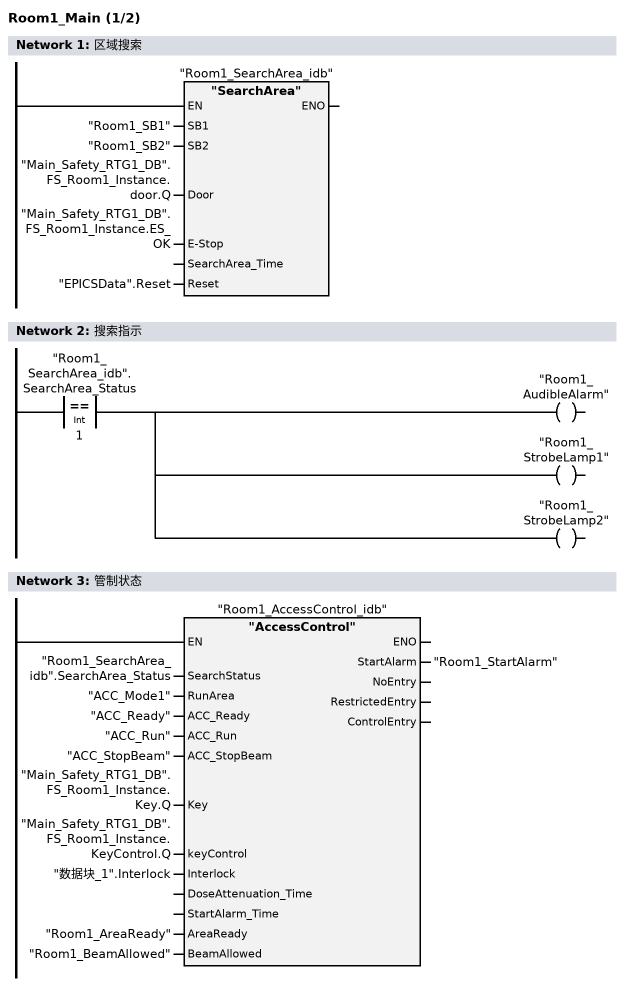
   RUNG wire#powerrail
      "Room1_SearchArea_idb"(SB1 := "Room1_SB1", SB2 := "Room1_SB2", Door := "Main_Safety_RTG1_DB".FS_Room1_Instance.door.Q, "E-Stop" := "Main_Safety_RTG1_DB".FS_Room1_Instance.ES_OK, SearchArea_Time :=, Reset := "EPICSData".Reset)
   END_RUNG
   // the same network as SCL:
   "Room1_SearchArea_idb"(SB1 := "Room1_SB1",   // "SearchArea"
                          SB2 := "Room1_SB2",
                          Door := "Main_Safety_RTG1_DB".FS_Room1_Instance.door.Q,
                          "E-Stop" := "Main_Safety_RTG1_DB".FS_Room1_Instance.ES_OK,
                          Reset := "EPICSData".Reset);
END_REGION

REGION Network 2: 搜索指示
   RUNG wire#powerrail
      { S7_Templates := "SrcType := Int" } EQ_Contact(in1 := "Room1_SearchArea_idb".SearchArea_Status, in2 := 1)
      wire#w1
      Coil( "Room1_AudibleAlarm" )
   END_RUNG
   RUNG wire#w1
      Coil( "Room1_StrobeLamp1" )
   END_RUNG
   RUNG wire#w1
      Coil( "Room1_StrobeLamp2" )
   END_RUNG
   // the same network as SCL:
   "Room1_AudibleAlarm" := "Room1_SearchArea_idb".SearchArea_Status = 1;
   "Room1_StrobeLamp1" := "Room1_AudibleAlarm";
   "Room1_StrobeLamp2" := "Room1_AudibleAlarm";
END_REGION

REGION Network 3: 管制状态
   RUNG wire#powerrail
      "Room1_AccessControl_idb"(SearchStatus := "Room1_SearchArea_idb".SearchArea_Status, RunArea := "ACC_Mode1", ACC_Ready := "ACC_Ready", ACC_Run := "ACC_Run", ACC_StopBeam := "ACC_StopBeam", Key := "Main_Safety_RTG1_DB".FS_Room1_Instance.Key.Q, keyControl := "Main_Safety_RTG1_DB".FS_Room1_Instance.KeyControl.Q, Interlock := "数据块_1".Interlock, DoseAttenuation_Time :=, StartAlarm_Time :=, AreaReady := "Room1_AreaReady", BeamAllowed := "Room1_BeamAllowed", StartAlarm => "Room1_StartAlarm", NoEntry =>, RestrictedEntry =>, ControlEntry =>)
   END_RUNG
   // the same network as SCL:
   "Room1_AccessControl_idb"(SearchStatus := "Room1_SearchArea_idb".SearchArea_Status,   // "AccessControl"
                           RunArea := "ACC_Mode1",
                           ACC_Ready := "ACC_Ready",
                           ACC_Run := "ACC_Run",
                           ACC_StopBeam := "ACC_StopBeam",
                           Key := "Main_Safety_RTG1_DB".FS_Room1_Instance.Key.Q,
                           keyControl := "Main_Safety_RTG1_DB".FS_Room1_Instance.KeyControl.Q,
                           Interlock := "数据块_1".Interlock,
                           AreaReady := "Room1_AreaReady",
                           BeamAllowed := "Room1_BeamAllowed",
                           StartAlarm => "Room1_StartAlarm");
END_REGION

REGION Network 4: 管制输出
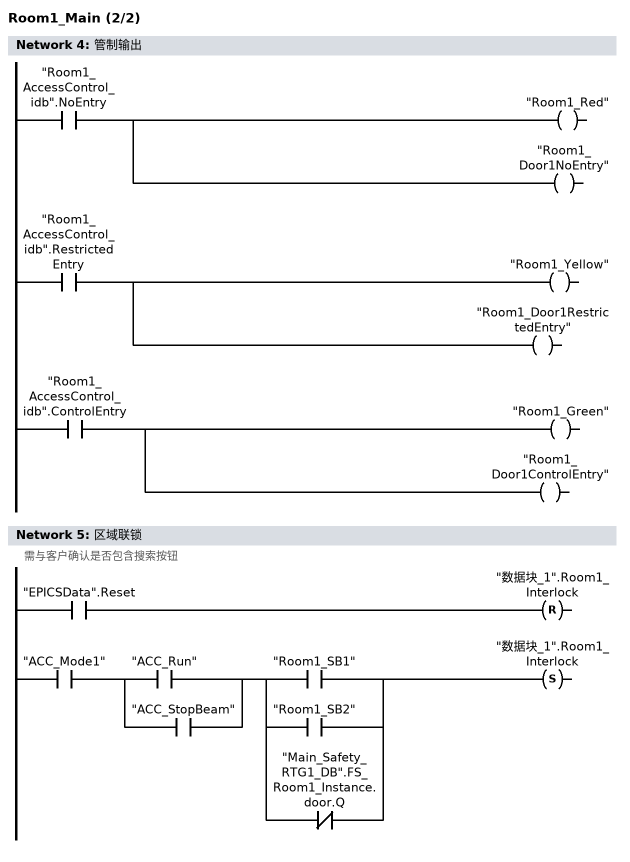
   RUNG wire#powerrail
      Contact( "Room1_AccessControl_idb".NoEntry )
      wire#w1
      Coil( "Room1_Red" )
   END_RUNG
   RUNG wire#w1
      Coil( "Room1_Door1NoEntry" )
   END_RUNG
   RUNG wire#powerrail
      Contact( "Room1_AccessControl_idb".RestrictedEntry )
      wire#w2
      Coil( "Room1_Yellow" )
   END_RUNG
   RUNG wire#w2
      Coil( "Room1_Door1RestrictedEntry" )
   END_RUNG
   RUNG wire#powerrail
      Contact( "Room1_AccessControl_idb".ControlEntry )
      wire#w3
      Coil( "Room1_Green" )
   END_RUNG
   RUNG wire#w3
      Coil( "Room1_Door1ControlEntry" )
   END_RUNG
   // the same network as SCL:
   "Room1_Red" := "Room1_AccessControl_idb".NoEntry;
   "Room1_Door1NoEntry" := "Room1_AccessControl_idb".NoEntry;
   "Room1_Yellow" := "Room1_AccessControl_idb".RestrictedEntry;
   "Room1_Door1RestrictedEntry" := "Room1_AccessControl_idb".RestrictedEntry;
   "Room1_Green" := "Room1_AccessControl_idb".ControlEntry;
   "Room1_Door1ControlEntry" := "Room1_AccessControl_idb".ControlEntry;
END_REGION

REGION Network 5: 区域联锁
   // 需与客户确认是否包含搜索按钮
   RUNG wire#powerrail
      Contact( "EPICSData".Reset )
      R_Coil( "数据块_1".Room1_Interlock )
   END_RUNG
   RUNG wire#powerrail
      Contact( "ACC_Mode1" )
      wire#w1
      Contact( "ACC_Run" )
      wire#w2
      Contact( "Room1_SB1" )
      wire#w3
      S_Coil( "数据块_1".Room1_Interlock )
   END_RUNG
   RUNG wire#w1
      Contact( "ACC_StopBeam" )
   END_RUNG wire#w2
   RUNG wire#w2
      Contact( "Room1_SB2" )
   END_RUNG wire#w3
   RUNG wire#w2
      I_Contact( "Main_Safety_RTG1_DB".FS_Room1_Instance.door.Q )
   END_RUNG wire#w3
   // the same network as SCL:
   IF "EPICSData".Reset THEN "数据块_1".Room1_Interlock := FALSE; END_IF;
   IF "ACC_Mode1" AND ("ACC_Run" OR "ACC_StopBeam") AND ("Room1_SB1" OR "Room1_SB2" OR NOT "Main_Safety_RTG1_DB".FS_Room1_Instance.door.Q) THEN
       "数据块_1".Room1_Interlock := TRUE;
   END_IF;
END_REGION
END_FUNCTION

FUNCTION "Room2_Main" : Void   // FC5, LAD
{ S7_Optimized_Access := 'TRUE' }
VERSION : 0.1
// stored: AutoNumber true, IsIECCheckEnabled false, SetENOAutomatically false, UDAEnableTagReadback false
BEGIN

REGION Network 1: 区域搜索
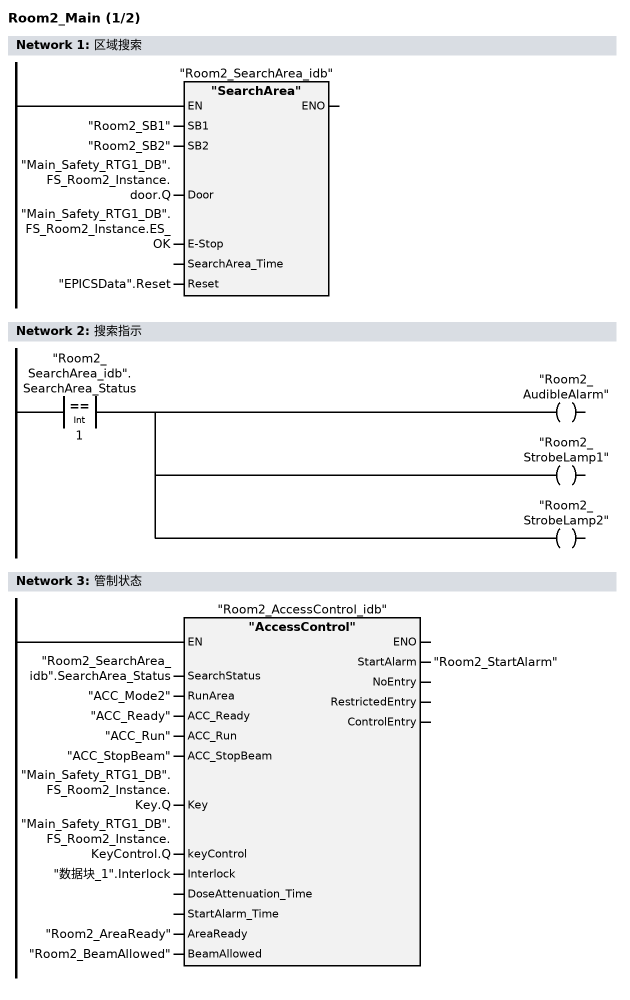
   RUNG wire#powerrail
      "Room2_SearchArea_idb"(SB1 := "Room2_SB1", SB2 := "Room2_SB2", Door := "Main_Safety_RTG1_DB".FS_Room2_Instance.door.Q, "E-Stop" := "Main_Safety_RTG1_DB".FS_Room2_Instance.ES_OK, SearchArea_Time :=, Reset := "EPICSData".Reset)
   END_RUNG
   // the same network as SCL:
   "Room2_SearchArea_idb"(SB1 := "Room2_SB1",   // "SearchArea"
                          SB2 := "Room2_SB2",
                          Door := "Main_Safety_RTG1_DB".FS_Room2_Instance.door.Q,
                          "E-Stop" := "Main_Safety_RTG1_DB".FS_Room2_Instance.ES_OK,
                          Reset := "EPICSData".Reset);
END_REGION

REGION Network 2: 搜索指示
   RUNG wire#powerrail
      { S7_Templates := "SrcType := Int" } EQ_Contact(in1 := "Room2_SearchArea_idb".SearchArea_Status, in2 := 1)
      wire#w1
      Coil( "Room2_AudibleAlarm" )
   END_RUNG
   RUNG wire#w1
      Coil( "Room2_StrobeLamp1" )
   END_RUNG
   RUNG wire#w1
      Coil( "Room2_StrobeLamp2" )
   END_RUNG
   // the same network as SCL:
   "Room2_AudibleAlarm" := "Room2_SearchArea_idb".SearchArea_Status = 1;
   "Room2_StrobeLamp1" := "Room2_AudibleAlarm";
   "Room2_StrobeLamp2" := "Room2_AudibleAlarm";
END_REGION

REGION Network 3: 管制状态
   RUNG wire#powerrail
      "Room2_AccessControl_idb"(SearchStatus := "Room2_SearchArea_idb".SearchArea_Status, RunArea := "ACC_Mode2", ACC_Ready := "ACC_Ready", ACC_Run := "ACC_Run", ACC_StopBeam := "ACC_StopBeam", Key := "Main_Safety_RTG1_DB".FS_Room2_Instance.Key.Q, keyControl := "Main_Safety_RTG1_DB".FS_Room2_Instance.KeyControl.Q, Interlock := "数据块_1".Interlock, DoseAttenuation_Time :=, StartAlarm_Time :=, AreaReady := "Room2_AreaReady", BeamAllowed := "Room2_BeamAllowed", StartAlarm => "Room2_StartAlarm", NoEntry =>, RestrictedEntry =>, ControlEntry =>)
   END_RUNG
   // the same network as SCL:
   "Room2_AccessControl_idb"(SearchStatus := "Room2_SearchArea_idb".SearchArea_Status,   // "AccessControl"
                           RunArea := "ACC_Mode2",
                           ACC_Ready := "ACC_Ready",
                           ACC_Run := "ACC_Run",
                           ACC_StopBeam := "ACC_StopBeam",
                           Key := "Main_Safety_RTG1_DB".FS_Room2_Instance.Key.Q,
                           keyControl := "Main_Safety_RTG1_DB".FS_Room2_Instance.KeyControl.Q,
                           Interlock := "数据块_1".Interlock,
                           AreaReady := "Room2_AreaReady",
                           BeamAllowed := "Room2_BeamAllowed",
                           StartAlarm => "Room2_StartAlarm");
END_REGION

REGION Network 4: 管制输出
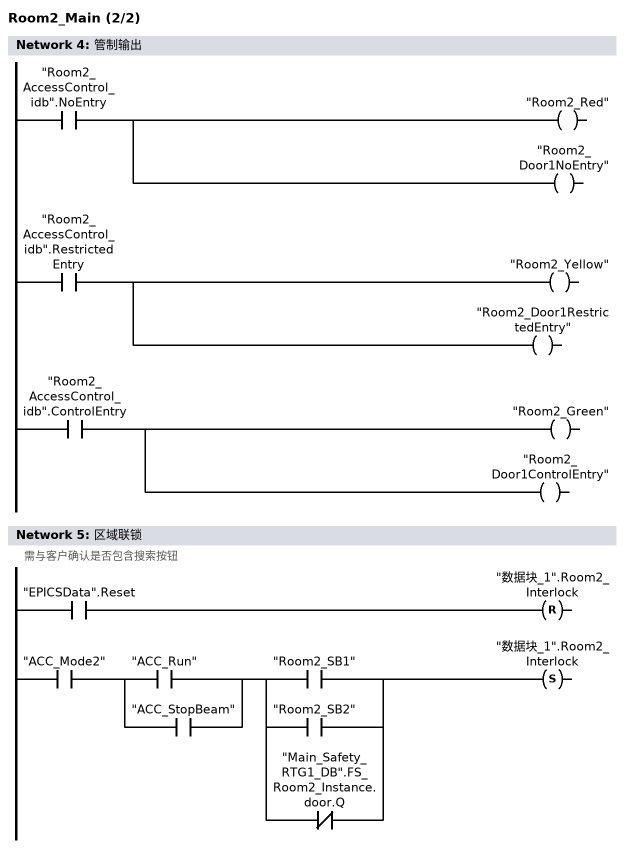
   RUNG wire#powerrail
      Contact( "Room2_AccessControl_idb".NoEntry )
      wire#w1
      Coil( "Room2_Red" )
   END_RUNG
   RUNG wire#w1
      Coil( "Room2_Door1NoEntry" )
   END_RUNG
   RUNG wire#powerrail
      Contact( "Room2_AccessControl_idb".RestrictedEntry )
      wire#w2
      Coil( "Room2_Yellow" )
   END_RUNG
   RUNG wire#w2
      Coil( "Room2_Door1RestrictedEntry" )
   END_RUNG
   RUNG wire#powerrail
      Contact( "Room2_AccessControl_idb".ControlEntry )
      wire#w3
      Coil( "Room2_Green" )
   END_RUNG
   RUNG wire#w3
      Coil( "Room2_Door1ControlEntry" )
   END_RUNG
   // the same network as SCL:
   "Room2_Red" := "Room2_AccessControl_idb".NoEntry;
   "Room2_Door1NoEntry" := "Room2_AccessControl_idb".NoEntry;
   "Room2_Yellow" := "Room2_AccessControl_idb".RestrictedEntry;
   "Room2_Door1RestrictedEntry" := "Room2_AccessControl_idb".RestrictedEntry;
   "Room2_Green" := "Room2_AccessControl_idb".ControlEntry;
   "Room2_Door1ControlEntry" := "Room2_AccessControl_idb".ControlEntry;
END_REGION

REGION Network 5: 区域联锁
   // 需与客户确认是否包含搜索按钮
   RUNG wire#powerrail
      Contact( "EPICSData".Reset )
      R_Coil( "数据块_1".Room2_Interlock )
   END_RUNG
   RUNG wire#powerrail
      Contact( "ACC_Mode2" )
      wire#w1
      Contact( "ACC_Run" )
      wire#w2
      Contact( "Room2_SB1" )
      wire#w3
      S_Coil( "数据块_1".Room2_Interlock )
   END_RUNG
   RUNG wire#w1
      Contact( "ACC_StopBeam" )
   END_RUNG wire#w2
   RUNG wire#w2
      Contact( "Room2_SB2" )
   END_RUNG wire#w3
   RUNG wire#w2
      I_Contact( "Main_Safety_RTG1_DB".FS_Room2_Instance.door.Q )
   END_RUNG wire#w3
   // the same network as SCL:
   IF "EPICSData".Reset THEN "数据块_1".Room2_Interlock := FALSE; END_IF;
   IF "ACC_Mode2" AND ("ACC_Run" OR "ACC_StopBeam") AND ("Room2_SB1" OR "Room2_SB2" OR NOT "Main_Safety_RTG1_DB".FS_Room2_Instance.door.Q) THEN
       "数据块_1".Room2_Interlock := TRUE;
   END_IF;
END_REGION
END_FUNCTION

FUNCTION "ACC_Main" : Void   // FC6, LAD
{ S7_Optimized_Access := 'TRUE' }
VERSION : 0.1
// stored: AutoNumber true, IsIECCheckEnabled false, SetENOAutomatically false, UDAEnableTagReadback false
BEGIN

REGION Network 1: 区域搜索
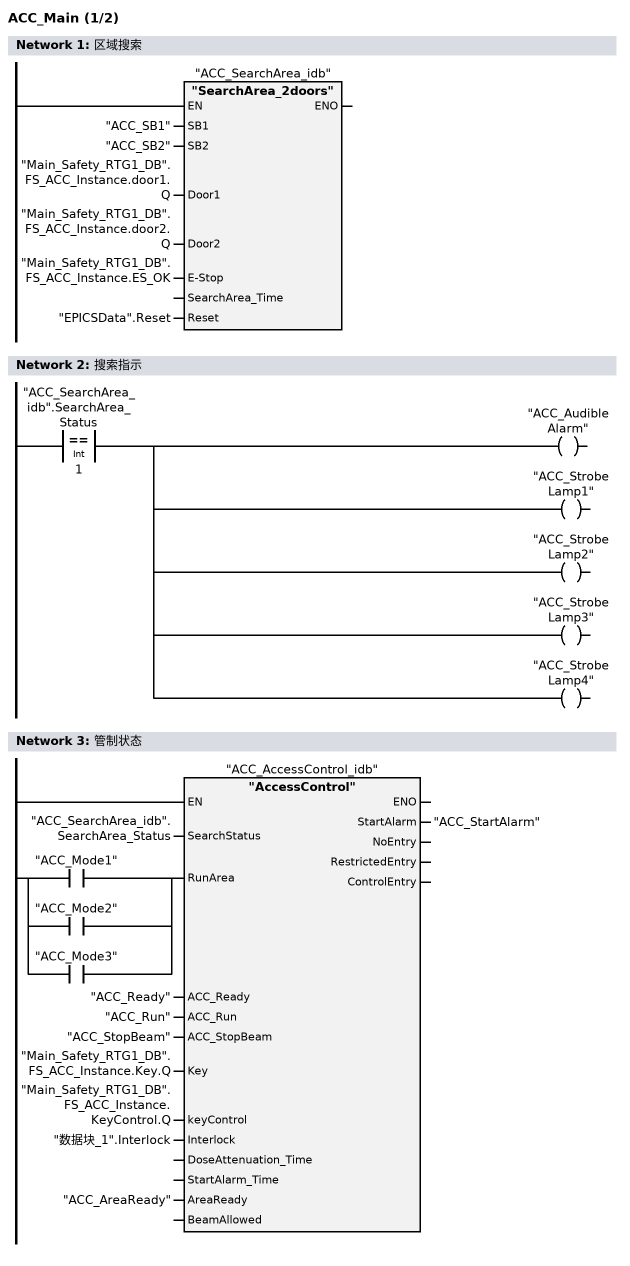
   RUNG wire#powerrail
      "ACC_SearchArea_idb"(SB1 := "ACC_SB1", SB2 := "ACC_SB2", Door1 := "Main_Safety_RTG1_DB".FS_ACC_Instance.door1.Q, Door2 := "Main_Safety_RTG1_DB".FS_ACC_Instance.door2.Q, "E-Stop" := "Main_Safety_RTG1_DB".FS_ACC_Instance.ES_OK, SearchArea_Time :=, Reset := "EPICSData".Reset)
   END_RUNG
   // the same network as SCL:
   "ACC_SearchArea_idb"(SB1 := "ACC_SB1",   // "SearchArea_2doors"
                        SB2 := "ACC_SB2",
                        Door1 := "Main_Safety_RTG1_DB".FS_ACC_Instance.door1.Q,
                        Door2 := "Main_Safety_RTG1_DB".FS_ACC_Instance.door2.Q,
                        "E-Stop" := "Main_Safety_RTG1_DB".FS_ACC_Instance.ES_OK,
                        Reset := "EPICSData".Reset);
END_REGION

REGION Network 2: 搜索指示
   RUNG wire#powerrail
      { S7_Templates := "SrcType := Int" } EQ_Contact(in1 := "ACC_SearchArea_idb".SearchArea_Status, in2 := 1)
      wire#w1
      Coil( "ACC_AudibleAlarm" )
   END_RUNG
   RUNG wire#w1
      Coil( "ACC_StrobeLamp1" )
   END_RUNG
   RUNG wire#w1
      Coil( "ACC_StrobeLamp2" )
   END_RUNG
   RUNG wire#w1
      Coil( "ACC_StrobeLamp3" )
   END_RUNG
   RUNG wire#w1
      Coil( "ACC_StrobeLamp4" )
   END_RUNG
   // the same network as SCL:
   "ACC_AudibleAlarm" := "ACC_SearchArea_idb".SearchArea_Status = 1;
   "ACC_StrobeLamp1" := "ACC_AudibleAlarm";
   "ACC_StrobeLamp2" := "ACC_AudibleAlarm";
   "ACC_StrobeLamp3" := "ACC_AudibleAlarm";
   "ACC_StrobeLamp4" := "ACC_AudibleAlarm";
END_REGION

REGION Network 3: 管制状态
   RUNG wire#powerrail
      "ACC_AccessControl_idb"(RunArea := wire#w1, SearchStatus := "ACC_SearchArea_idb".SearchArea_Status, ACC_Ready := "ACC_Ready", ACC_Run := "ACC_Run", ACC_StopBeam := "ACC_StopBeam", Key := "Main_Safety_RTG1_DB".FS_ACC_Instance.Key.Q, keyControl := "Main_Safety_RTG1_DB".FS_ACC_Instance.KeyControl.Q, Interlock := "数据块_1".Interlock, DoseAttenuation_Time :=, StartAlarm_Time :=, AreaReady := "ACC_AreaReady", BeamAllowed :=, StartAlarm => "ACC_StartAlarm", NoEntry =>, RestrictedEntry =>, ControlEntry =>)
   END_RUNG
   RUNG wire#powerrail
      Contact( "ACC_Mode1" )
   END_RUNG wire#w1
   RUNG wire#powerrail
      Contact( "ACC_Mode2" )
   END_RUNG wire#w1
   RUNG wire#powerrail
      Contact( "ACC_Mode3" )
   END_RUNG wire#w1
   // the same network as SCL:
   "ACC_AccessControl_idb"(SearchStatus := "ACC_SearchArea_idb".SearchArea_Status,   // "AccessControl"
                           RunArea := "ACC_Mode1" OR "ACC_Mode2" OR "ACC_Mode3",
                           ACC_Ready := "ACC_Ready",
                           ACC_Run := "ACC_Run",
                           ACC_StopBeam := "ACC_StopBeam",
                           Key := "Main_Safety_RTG1_DB".FS_ACC_Instance.Key.Q,
                           keyControl := "Main_Safety_RTG1_DB".FS_ACC_Instance.KeyControl.Q,
                           Interlock := "数据块_1".Interlock,
                           AreaReady := "ACC_AreaReady",
                           StartAlarm => "ACC_StartAlarm");
END_REGION

REGION Network 4: 管制输出
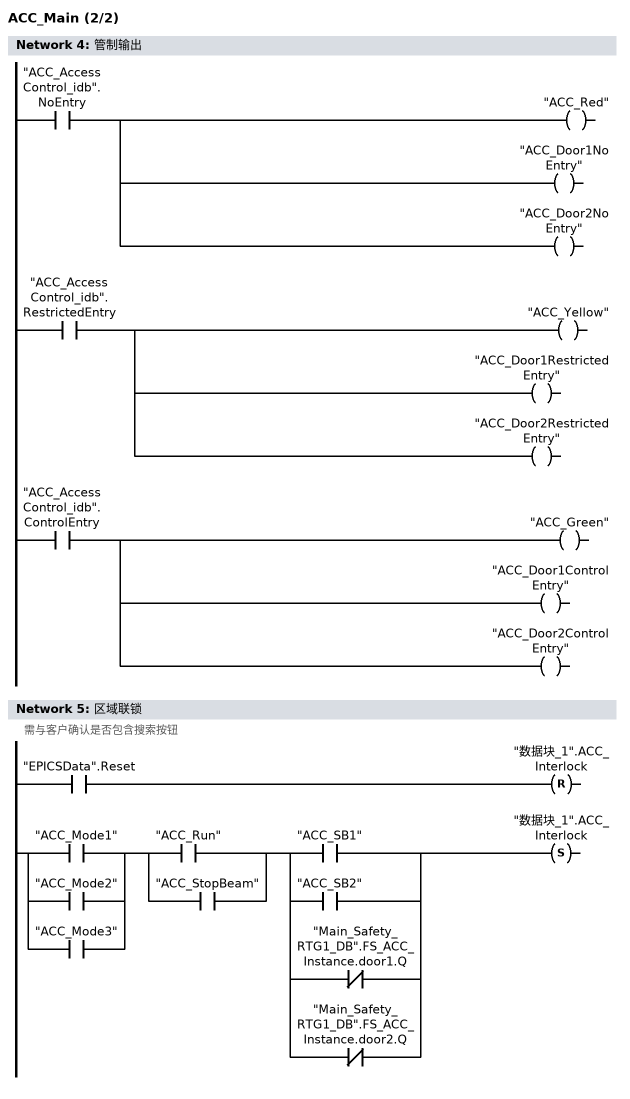
   RUNG wire#powerrail
      Contact( "ACC_AccessControl_idb".NoEntry )
      wire#w1
      Coil( "ACC_Red" )
   END_RUNG
   RUNG wire#w1
      Coil( "ACC_Door1NoEntry" )
   END_RUNG
   RUNG wire#w1
      Coil( "ACC_Door2NoEntry" )
   END_RUNG
   RUNG wire#powerrail
      Contact( "ACC_AccessControl_idb".RestrictedEntry )
      wire#w2
      Coil( "ACC_Yellow" )
   END_RUNG
   RUNG wire#w2
      Coil( "ACC_Door1RestrictedEntry" )
   END_RUNG
   RUNG wire#w2
      Coil( "ACC_Door2RestrictedEntry" )
   END_RUNG
   RUNG wire#powerrail
      Contact( "ACC_AccessControl_idb".ControlEntry )
      wire#w3
      Coil( "ACC_Green" )
   END_RUNG
   RUNG wire#w3
      Coil( "ACC_Door1ControlEntry" )
   END_RUNG
   RUNG wire#w3
      Coil( "ACC_Door2ControlEntry" )
   END_RUNG
   // the same network as SCL:
   "ACC_Red" := "ACC_AccessControl_idb".NoEntry;
   "ACC_Door1NoEntry" := "ACC_AccessControl_idb".NoEntry;
   "ACC_Door2NoEntry" := "ACC_AccessControl_idb".NoEntry;
   "ACC_Yellow" := "ACC_AccessControl_idb".RestrictedEntry;
   "ACC_Door1RestrictedEntry" := "ACC_AccessControl_idb".RestrictedEntry;
   "ACC_Door2RestrictedEntry" := "ACC_AccessControl_idb".RestrictedEntry;
   "ACC_Green" := "ACC_AccessControl_idb".ControlEntry;
   "ACC_Door1ControlEntry" := "ACC_AccessControl_idb".ControlEntry;
   "ACC_Door2ControlEntry" := "ACC_AccessControl_idb".ControlEntry;
END_REGION

REGION Network 5: 区域联锁
   // 需与客户确认是否包含搜索按钮
   RUNG wire#powerrail
      Contact( "EPICSData".Reset )
      R_Coil( "数据块_1".ACC_Interlock )
   END_RUNG
   RUNG wire#powerrail
      Contact( "ACC_Mode1" )
      wire#w1
      Contact( "ACC_Run" )
      wire#w2
      Contact( "ACC_SB1" )
      wire#w3
      S_Coil( "数据块_1".ACC_Interlock )
   END_RUNG
   RUNG wire#powerrail
      Contact( "ACC_Mode2" )
   END_RUNG wire#w1
   RUNG wire#powerrail
      Contact( "ACC_Mode3" )
   END_RUNG wire#w1
   RUNG wire#w1
      Contact( "ACC_StopBeam" )
   END_RUNG wire#w2
   RUNG wire#w2
      Contact( "ACC_SB2" )
   END_RUNG wire#w3
   RUNG wire#w2
      I_Contact( "Main_Safety_RTG1_DB".FS_ACC_Instance.door1.Q )
   END_RUNG wire#w3
   RUNG wire#w2
      I_Contact( "Main_Safety_RTG1_DB".FS_ACC_Instance.door2.Q )
   END_RUNG wire#w3
   // the same network as SCL:
   IF "EPICSData".Reset THEN "数据块_1".ACC_Interlock := FALSE; END_IF;
   IF ("ACC_Mode1" OR "ACC_Mode2" OR "ACC_Mode3") AND ("ACC_Run" OR "ACC_StopBeam") AND ("ACC_SB1" OR "ACC_SB2" OR NOT "Main_Safety_RTG1_DB".FS_ACC_Instance.door1.Q OR NOT "Main_Safety_RTG1_DB".FS_ACC_Instance.door2.Q) THEN
       "数据块_1".ACC_Interlock := TRUE;
   END_IF;
END_REGION
END_FUNCTION

FUNCTION "VerticalBeam_Main" : Void   // FC7, LAD
{ S7_Optimized_Access := 'TRUE' }
VERSION : 0.1
// stored: AutoNumber true, IsIECCheckEnabled false, SetENOAutomatically false, UDAEnableTagReadback false
BEGIN

REGION Network 1: 区域搜索
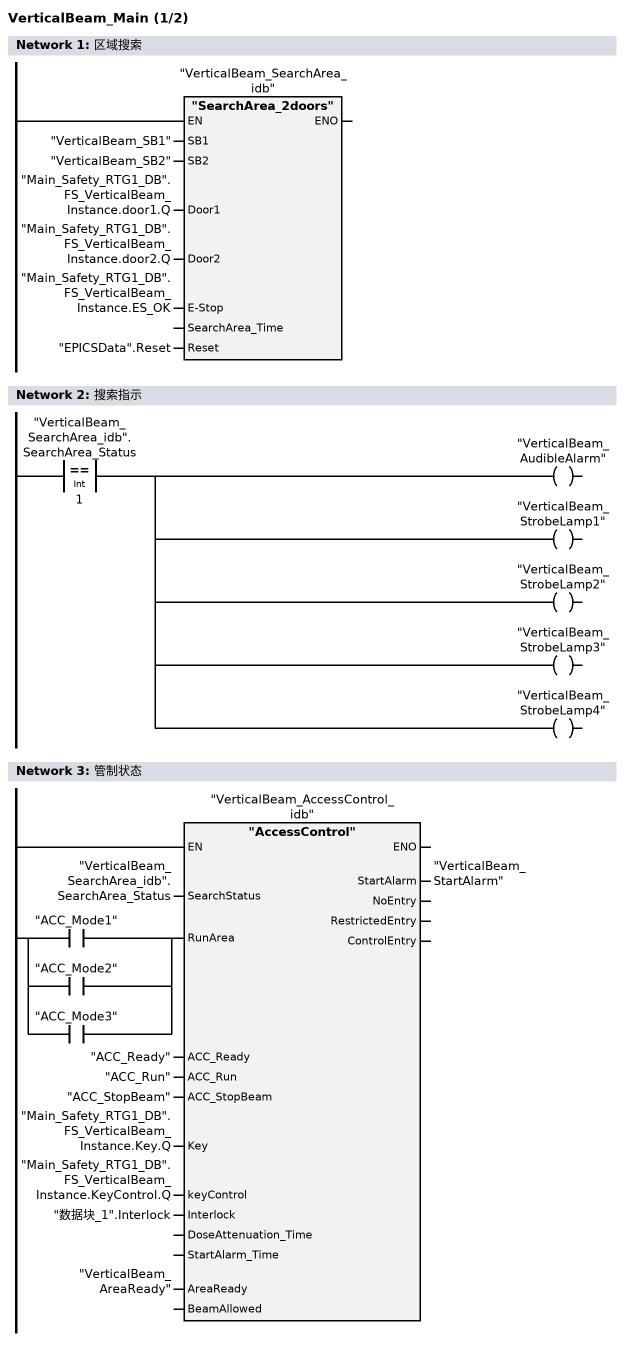
   RUNG wire#powerrail
      "VerticalBeam_SearchArea_idb"(SB1 := "VerticalBeam_SB1", SB2 := "VerticalBeam_SB2", Door1 := "Main_Safety_RTG1_DB".FS_VerticalBeam_Instance.door1.Q, Door2 := "Main_Safety_RTG1_DB".FS_VerticalBeam_Instance.door2.Q, "E-Stop" := "Main_Safety_RTG1_DB".FS_VerticalBeam_Instance.ES_OK, SearchArea_Time :=, Reset := "EPICSData".Reset)
   END_RUNG
   // the same network as SCL:
   "VerticalBeam_SearchArea_idb"(SB1 := "VerticalBeam_SB1",   // "SearchArea_2doors"
                           SB2 := "VerticalBeam_SB2",
                           Door1 := "Main_Safety_RTG1_DB".FS_VerticalBeam_Instance.door1.Q,
                           Door2 := "Main_Safety_RTG1_DB".FS_VerticalBeam_Instance.door2.Q,
                           "E-Stop" := "Main_Safety_RTG1_DB".FS_VerticalBeam_Instance.ES_OK,
                           Reset := "EPICSData".Reset);
END_REGION

REGION Network 2: 搜索指示
   RUNG wire#powerrail
      { S7_Templates := "SrcType := Int" } EQ_Contact(in1 := "VerticalBeam_SearchArea_idb".SearchArea_Status, in2 := 1)
      wire#w1
      Coil( "VerticalBeam_AudibleAlarm" )
   END_RUNG
   RUNG wire#w1
      Coil( "VerticalBeam_StrobeLamp1" )
   END_RUNG
   RUNG wire#w1
      Coil( "VerticalBeam_StrobeLamp2" )
   END_RUNG
   RUNG wire#w1
      Coil( "VerticalBeam_StrobeLamp3" )
   END_RUNG
   RUNG wire#w1
      Coil( "VerticalBeam_StrobeLamp4" )
   END_RUNG
   // the same network as SCL:
   "VerticalBeam_AudibleAlarm" := "VerticalBeam_SearchArea_idb".SearchArea_Status = 1;
   "VerticalBeam_StrobeLamp1" := "VerticalBeam_AudibleAlarm";
   "VerticalBeam_StrobeLamp2" := "VerticalBeam_AudibleAlarm";
   "VerticalBeam_StrobeLamp3" := "VerticalBeam_AudibleAlarm";
   "VerticalBeam_StrobeLamp4" := "VerticalBeam_AudibleAlarm";
END_REGION

REGION Network 3: 管制状态
   RUNG wire#powerrail
      "VerticalBeam_AccessControl_idb"(RunArea := wire#w1, SearchStatus := "VerticalBeam_SearchArea_idb".SearchArea_Status, ACC_Ready := "ACC_Ready", ACC_Run := "ACC_Run", ACC_StopBeam := "ACC_StopBeam", Key := "Main_Safety_RTG1_DB".FS_VerticalBeam_Instance.Key.Q, keyControl := "Main_Safety_RTG1_DB".FS_VerticalBeam_Instance.KeyControl.Q, Interlock := "数据块_1".Interlock, DoseAttenuation_Time :=, StartAlarm_Time :=, AreaReady := "VerticalBeam_AreaReady", BeamAllowed :=, StartAlarm => "VerticalBeam_StartAlarm", NoEntry =>, RestrictedEntry =>, ControlEntry =>)
   END_RUNG
   RUNG wire#powerrail
      Contact( "ACC_Mode1" )
   END_RUNG wire#w1
   RUNG wire#powerrail
      Contact( "ACC_Mode2" )
   END_RUNG wire#w1
   RUNG wire#powerrail
      Contact( "ACC_Mode3" )
   END_RUNG wire#w1
   // the same network as SCL:
   "VerticalBeam_AccessControl_idb"(SearchStatus := "VerticalBeam_SearchArea_idb".SearchArea_Status,   // "AccessControl"
                           RunArea := "ACC_Mode1" OR "ACC_Mode2" OR "ACC_Mode3",
                           ACC_Ready := "ACC_Ready",
                           ACC_Run := "ACC_Run",
                           ACC_StopBeam := "ACC_StopBeam",
                           Key := "Main_Safety_RTG1_DB".FS_VerticalBeam_Instance.Key.Q,
                           keyControl := "Main_Safety_RTG1_DB".FS_VerticalBeam_Instance.KeyControl.Q,
                           Interlock := "数据块_1".Interlock,
                           AreaReady := "VerticalBeam_AreaReady",
                           StartAlarm => "VerticalBeam_StartAlarm");
END_REGION

REGION Network 4: 管制输出
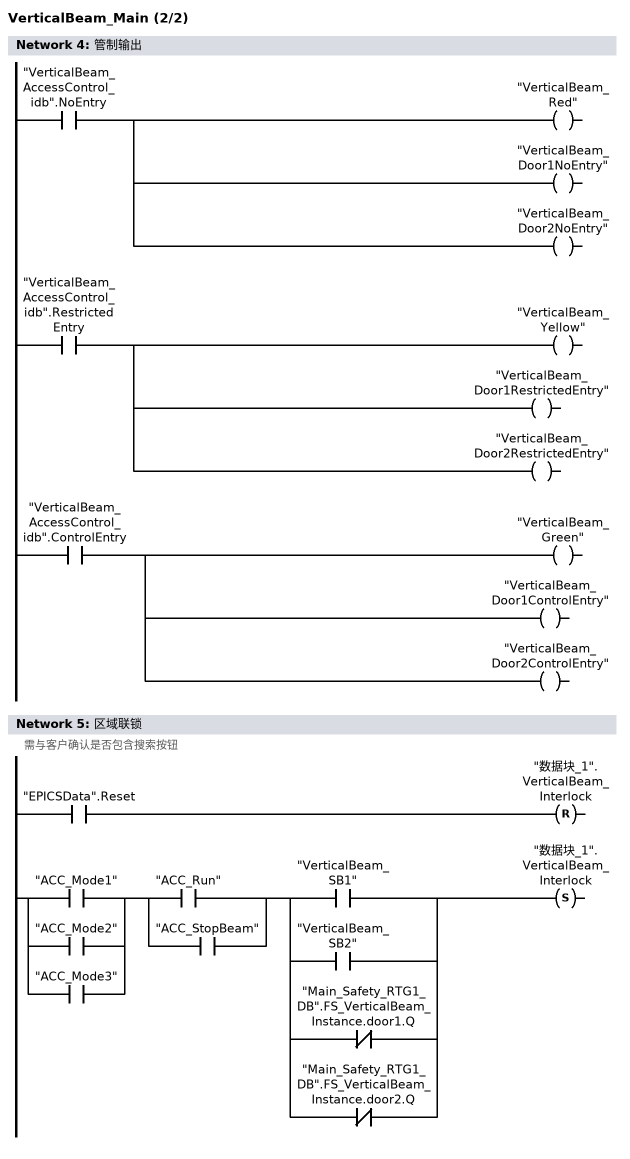
   RUNG wire#powerrail
      Contact( "VerticalBeam_AccessControl_idb".NoEntry )
      wire#w1
      Coil( "VerticalBeam_Red" )
   END_RUNG
   RUNG wire#w1
      Coil( "VerticalBeam_Door1NoEntry" )
   END_RUNG
   RUNG wire#w1
      Coil( "VerticalBeam_Door2NoEntry" )
   END_RUNG
   RUNG wire#powerrail
      Contact( "VerticalBeam_AccessControl_idb".RestrictedEntry )
      wire#w2
      Coil( "VerticalBeam_Yellow" )
   END_RUNG
   RUNG wire#w2
      Coil( "VerticalBeam_Door1RestrictedEntry" )
   END_RUNG
   RUNG wire#w2
      Coil( "VerticalBeam_Door2RestrictedEntry" )
   END_RUNG
   RUNG wire#powerrail
      Contact( "VerticalBeam_AccessControl_idb".ControlEntry )
      wire#w3
      Coil( "VerticalBeam_Green" )
   END_RUNG
   RUNG wire#w3
      Coil( "VerticalBeam_Door1ControlEntry" )
   END_RUNG
   RUNG wire#w3
      Coil( "VerticalBeam_Door2ControlEntry" )
   END_RUNG
   // the same network as SCL:
   "VerticalBeam_Red" := "VerticalBeam_AccessControl_idb".NoEntry;
   "VerticalBeam_Door1NoEntry" := "VerticalBeam_AccessControl_idb".NoEntry;
   "VerticalBeam_Door2NoEntry" := "VerticalBeam_AccessControl_idb".NoEntry;
   "VerticalBeam_Yellow" := "VerticalBeam_AccessControl_idb".RestrictedEntry;
   "VerticalBeam_Door1RestrictedEntry" := "VerticalBeam_AccessControl_idb".RestrictedEntry;
   "VerticalBeam_Door2RestrictedEntry" := "VerticalBeam_AccessControl_idb".RestrictedEntry;
   "VerticalBeam_Green" := "VerticalBeam_AccessControl_idb".ControlEntry;
   "VerticalBeam_Door1ControlEntry" := "VerticalBeam_AccessControl_idb".ControlEntry;
   "VerticalBeam_Door2ControlEntry" := "VerticalBeam_AccessControl_idb".ControlEntry;
END_REGION

REGION Network 5: 区域联锁
   // 需与客户确认是否包含搜索按钮
   RUNG wire#powerrail
      Contact( "EPICSData".Reset )
      R_Coil( "数据块_1".VerticalBeam_Interlock )
   END_RUNG
   RUNG wire#powerrail
      Contact( "ACC_Mode1" )
      wire#w1
      Contact( "ACC_Run" )
      wire#w2
      Contact( "VerticalBeam_SB1" )
      wire#w3
      S_Coil( "数据块_1".VerticalBeam_Interlock )
   END_RUNG
   RUNG wire#powerrail
      Contact( "ACC_Mode2" )
   END_RUNG wire#w1
   RUNG wire#powerrail
      Contact( "ACC_Mode3" )
   END_RUNG wire#w1
   RUNG wire#w1
      Contact( "ACC_StopBeam" )
   END_RUNG wire#w2
   RUNG wire#w2
      Contact( "VerticalBeam_SB2" )
   END_RUNG wire#w3
   RUNG wire#w2
      I_Contact( "Main_Safety_RTG1_DB".FS_VerticalBeam_Instance.door1.Q )
   END_RUNG wire#w3
   RUNG wire#w2
      I_Contact( "Main_Safety_RTG1_DB".FS_VerticalBeam_Instance.door2.Q )
   END_RUNG wire#w3
   // the same network as SCL:
   IF "EPICSData".Reset THEN "数据块_1".VerticalBeam_Interlock := FALSE; END_IF;
   IF ("ACC_Mode1" OR "ACC_Mode2" OR "ACC_Mode3") AND ("ACC_Run" OR "ACC_StopBeam") AND ("VerticalBeam_SB1" OR "VerticalBeam_SB2" OR NOT "Main_Safety_RTG1_DB".FS_VerticalBeam_Instance.door1.Q OR NOT "Main_Safety_RTG1_DB".FS_VerticalBeam_Instance.door2.Q) THEN
       "数据块_1".VerticalBeam_Interlock := TRUE;
   END_IF;
END_REGION
END_FUNCTION

FUNCTION "TCS" : Void   // FC3, LAD
{ S7_Optimized_Access := 'TRUE' }
VERSION : 0.1
// stored: AutoNumber true, IsIECCheckEnabled false, SetENOAutomatically false, UDAEnableTagReadback false
BEGIN

REGION Network 1
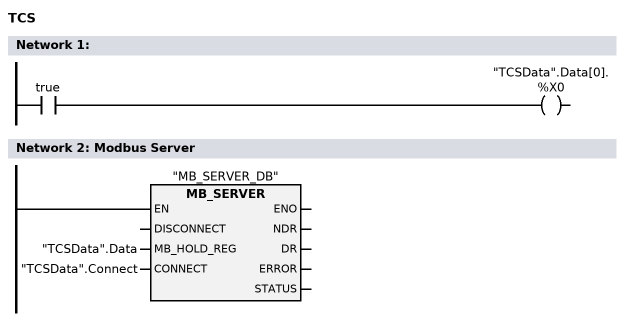
   RUNG wire#powerrail
      Contact( true )
      Coil( "TCSData".Data[0].%X0 )
   END_RUNG
   // the same network as SCL:
   "TCSData".Data[0].%X0 := true;
END_REGION

REGION Network 2: Modbus Server
   RUNG wire#powerrail
      "MB_SERVER_DB".MB_SERVER(DISCONNECT :=, MB_HOLD_REG := "TCSData".Data, CONNECT := "TCSData".Connect, NDR =>, DR =>, ERROR =>, STATUS =>)
   END_RUNG
   // the same network as SCL:
   "MB_SERVER_DB"(MB_HOLD_REG := "TCSData".Data, CONNECT := "TCSData".Connect);   // MB_SERVER
END_REGION
END_FUNCTION

DATA_BLOCK "MB_SERVER_DB"   // DB1
// stored: AutoNumber true, DBAccessibleFromOPCUA true, InstanceOfName MB_SERVER, OfSystemLibElement MB_SERVER, OfSystemLibVersion 5.3
"MB_SERVER"
   // VAR_INPUT
   //    DISCONNECT { ExternalVisible := 'False'} : Bool;
   // END_VAR
   // VAR_OUTPUT
   //    NDR { ExternalVisible := 'False'} : Bool;
   //    DR { ExternalVisible := 'False'} : Bool;
   //    ERROR { ExternalVisible := 'False'} : Bool;
   //    STATUS { ExternalVisible := 'False'} : Word;
   // END_VAR
   // VAR_IN_OUT
   //    MB_HOLD_REG : Variant;
   //    CONNECT : Variant;
   // END_VAR
   // VAR
   //    TCON { S7_SetPoint := 'True'} : TCON;
   //    TSEND { S7_SetPoint := 'True'} : TSEND;
   //    TRCV { S7_SetPoint := 'True'} : TRCV;
   //    TDIAG { S7_SetPoint := 'True'} : T_DIAG;
   //    TRESET { S7_SetPoint := 'True'} : T_RESET;
   //    TDISCON { S7_SetPoint := 'True'} : TDISCON;
   //    TDIAG_Status { S7_SetPoint := 'True'} : TDiag_Status;
   //    HR_Start_Offset : Word;
   //    QB_Start : UInt;
   //    QB_Count : UInt;
   //    QB_Read_Start : UInt;
   //    QB_Read_Count : UInt;
   //    IB_Read_Start : UInt;
   //    IB_Read_Count : UInt;
   //    Success_Count : Word;
   //    Request_Count : Word;
   //    Xmt_Rcv_Count : Word;
   //    Server_Message_Count : Word;
   //    Exception_Count : Word;
   //    Connected : Bool;
   //    Connection_ID { ExternalVisible := 'False'} : Word;
   //    MB_State : Word;
   //    TEMP_DATA { ExternalVisible := 'False'} : Array[0..262] of Byte;
   //    Data_Area_Array { S7_SetPoint := 'True'} : Array[1..8] of MB_DataArea;
   //    NDR_immediate : Bool;
   //    DR_immediate : Bool;
   //    BytesReceived : UDInt;
   //    overflow_buffer : Array[0..262] of Byte;
   //    overflow_size_bytes : UInt;
   // END_VAR
BEGIN
END_DATA_BLOCK

DATA_BLOCK "Main_Safety_RTG1_DB"   // DB1, F_DB
NAME : FUSI
VERSION : 0.1
// stored: AutoNumber true, DBAccessibleFromOPCUA true, InstanceOfName Main_Safety_RTG1, InstanceOfType FB
"Main_Safety_RTG1"
BEGIN
END_DATA_BLOCK

DATA_BLOCK "Room1_AccessControl_idb"   // DB9
VERSION : 0.1
// stored: AutoNumber true, DBAccessibleFromOPCUA true, InstanceOfName AccessControl, InstanceOfType FB
"AccessControl"
BEGIN
END_DATA_BLOCK

DATA_BLOCK "Room1_SearchArea_idb"   // DB6
VERSION : 0.1
// stored: AutoNumber true, DBAccessibleFromOPCUA true, InstanceOfName SearchArea, InstanceOfType FB
"SearchArea"
BEGIN
END_DATA_BLOCK

DATA_BLOCK "Room2_AccessControl_idb"   // DB10
VERSION : 0.1
// stored: AutoNumber true, DBAccessibleFromOPCUA true, InstanceOfName AccessControl, InstanceOfType FB
"AccessControl"
BEGIN
END_DATA_BLOCK

DATA_BLOCK "Room2_SearchArea_idb"   // DB7
VERSION : 0.1
// stored: AutoNumber true, DBAccessibleFromOPCUA true, InstanceOfName SearchArea, InstanceOfType FB
"SearchArea"
BEGIN
END_DATA_BLOCK

DATA_BLOCK "ACC_AccessControl_idb"   // DB12
VERSION : 0.1
// stored: AutoNumber true, DBAccessibleFromOPCUA true, InstanceOfName AccessControl, InstanceOfType FB
"AccessControl"
BEGIN
END_DATA_BLOCK

DATA_BLOCK "ACC_SearchArea_idb"   // DB11
VERSION : 0.1
// stored: AutoNumber true, DBAccessibleFromOPCUA true, InstanceOfName SearchArea_2doors, InstanceOfType FB
"SearchArea_2doors"
BEGIN
END_DATA_BLOCK

DATA_BLOCK "VerticalBeam_AccessControl_idb"   // DB14
VERSION : 0.1
// stored: AutoNumber true, DBAccessibleFromOPCUA true, InstanceOfName AccessControl, InstanceOfType FB
"AccessControl"
BEGIN
END_DATA_BLOCK

DATA_BLOCK "VerticalBeam_SearchArea_idb"   // DB13
VERSION : 0.1
// stored: AutoNumber true, DBAccessibleFromOPCUA true, InstanceOfName SearchArea_2doors, InstanceOfType FB
"SearchArea_2doors"
BEGIN
END_DATA_BLOCK
